//{{V2}}
FUNCTION FC15
TITLE= <Beschreibung der FC>


AUTHOR:nb
FAMILY:nb
NAME:nb
VERSION:1.0


VAR_INPUT
END_VAR

VAR_OUTPUT
END_VAR

VAR_IN_OUT
END_VAR

VAR_TEMP
END_VAR
BEGIN

NETWORK
TITLE=   <Ueberschrift von Netzwerk>
//{{a}}




END_FUNCTION
